// TIA Portal V17 export
// export: Created 2024-09-02T12:50:18.2983869Z, ExportSetting WithDefaults, DisplayName Totally Integrated Automation Portal, DisplayVersion V17, DisplayName TIA Portal Openness, DisplayVersion V17, DisplayName TIA Portal Version Control Interface, DisplayVersion V17, DisplayName STEP 7 Professional, DisplayVersion V17, DisplayName STEP 7 Safety, DisplayVersion V17, DisplayName WinCC Professional, DisplayVersion V17
DATA_BLOCK "LTLL_ManualGraphConfig_OP70"   // DB463
TITLE = LTLL_ManualGraphConfig
{ S7_Optimized_Access := 'TRUE'; DB_Accessible_From_OPC_UA := 'FALSE' }
AUTHOR : Siemens
FAMILY : HMI_Lite
NAME : LTLL_ManualGraphConfig
VERSION : 8.10
// stored: AutoNumber true, DBAccessibleFromOPCUA false, InstanceOfName LTLL_typeManualGraphConfig, InstanceOfType UDT, IsOnlyStoredInLoadMemory false, IsWriteProtectedInAS false
"LTLL_typeManualGraphConfig"
   // VAR
   //    row { S7_SetPoint := 'True'} : Array[1..348] of "LTLL_typeGraphConfigRow";
   // END_VAR
BEGIN
   row[1..2].left.dbInstanceName := WSTRING#'"DI_Hand_Schrittkette"';
   row[7..8].left.dbInstanceName := WSTRING#'"InstGraph1"';
   row[1].left.stepNumber := 1;
   row[2].left.stepNumber := 3;
   row[7].left.stepNumber := 1;
   row[8].left.stepNumber := 3;
   row[1..2].right.dbInstanceName := WSTRING#'"DI_Hand_Schrittkette"';
   row[7].right.dbInstanceName := WSTRING#'"InstGraph1"';
   row[1].right.stepNumber := 2;
   row[2].right.stepNumber := 4;
   row[7].right.stepNumber := 2;
END_DATA_BLOCK
